FUNCTION_BLOCK PUBLIC FB_HeatingZone
VAR_INPUT
	mxEnableHeating 				: BOOL;
	mxReset							: BOOL;
	mxEmergency						: BOOL;
	mxDoorsOpened					: BOOL;
END_VAR
VAR_OUTPUT
	mxErrorInit						: BOOL;
	mxErrorStopInPos				: BOOL;
	Errors							: ST_HeatingZoneErrors;
END_VAR
VAR

	qxPWMOut1 AT%Q*					: BOOL;
	qxPWMOut2 AT%Q*					: BOOL;
	qxPWMOut3 AT%Q*					: BOOL;
	ixThermal AT%I*					: BOOL;
	
	FT_EnableHeating				:F_Trig;	

	FB_Heating_Controller			: FB_PIDCtrl;
	FB_PID							: FB_PID_CP;
	FB_PWM							: FB_CTRL_PWM_OUT;
	FB_Temperature					: FB_AnalogInPT100;
	RT_EmStop						: R_TRIG;
	FT_EmStop						: F_TRIG;
	ControlMode						: E_CTRL_MODE;
	RT_ActivateHeating				: R_TRIG;
	RT_TempError					: R_TRIG;
	
	T_TempBelowSetpoint				: TON;
	SR_TempBelowSetpoint			: SR;
	T_TempAboveSetpoint				: TON;
	SR_TempAboveSetpoint			: SR;
	T_TimeInAutomode				: TON;

	T_HeatingStarted				: TON;

	SR_PT100_Loose					: SR;
	SR_PT100_WireBreakActive		: SR;
	SR_PT100_HasWrongPosition		: SR;
	SR_PT100_NotInserted			: SR;
	SR_PT100_ConnectorNotConnected	: SR;
	SR_PT100_ResistorFound	: SR;
	
	T_PT100_CheckTemperatures		: TON;
	mxIncreasedTemperatureNonActive	: BOOL;
	mxNoIncreaseTemperatureActive	: BOOL;
	OldTemperature					: REAL;
	
	T_PT100_HasWrongPosition		: Ton;
	FT_ActivateHeating: F_TRIG;
	SR_PT100_EnabledZoneWithoutProperPt100: SR;
	SR_TemperatureWayTooHigh: SR;
	
	Setpoint 			 	: REAL;
	TemperatureDifference	: REAL;
	SetpointStep		 	: REAL;
	ActStepNr            	: INT;
	ActTempMemory 			: REAL;
	PIDsetpoint				: REAL;
	mxSetpointReached		: BOOL;
	T_TempAtSetpointDelayNextStep	: TON;
	RT_StartHeatingInSteps			: R_TRIG;
	HeatingInSteps					: BOOL;
	RT_StopHeatingInSteps: R_TRIG;
	RT_DoorOpened: R_TRIG;
	FT_DoorOpened: F_TRIG;
	RT_HeatingPIDON: R_TRIG;
	FT_HeatingPIDON: F_TRIG;
	RT_SetPointChanged: R_TRIG;
	OldSetpoint: REAL; 
	SR_TemperatureTooHighWarning: SR;
END_VAR
VAR_IN_OUT
	MachParameters					: ST_HeatingZone;
END_VAR

DetermineSetpoint();
Error();
Objects();

RT_ActivateHeating(CLK:=MachParameters.mxZoneActive);
T_HeatingStarted(IN:=, PT:=T#10M);

RT_HeatingPIDON(CLK:=FB_Heating_Controller.PID_ON);
FT_HeatingPIDON(CLK:=FB_Heating_Controller.PID_ON);

FB_Heating_Controller.PID_ON := mxEnableHeating AND MachParameters.mxZoneActive AND NOT mxEmergency AND NOT FB_Temperature.Error;

// Start heating "started" timer when heating switches on
IF RT_HeatingPIDON.Q THEN
	T_HeatingStarted.IN := TRUE;
END_IF

IF NOT FB_Heating_Controller.PID_ON THEN
	T_HeatingStarted.IN :=FALSE;
END_IF

// Autoreset the PWM controller when a error occures
IF FB_PWM.bError AND (ControlMode = eCTRL_MODE_ACTIVE) THEN
	Controlmode := eCTRL_MODE_RESET;
ELSE
	ControlMode := eCTRL_MODE_ACTIVE;
END_IF

OldSetpoint := MachParameters.PIDTempZone.SP_AUTO;

ACTION DetermineSetpoint:
// because of enormous overshoots, the setpoint of the PID is scaled up during startup
// and cut into smaller heating steps. For example when a 180 degree setpoint is set in the HMI
// And the number of warmingsteps is set to 10. The PID first gets a setpoint of: 180/10 * 1
// When the setpoint is reached the timer "SetpointReached" starts counting. When this timer
// is elapsed the next set is set into the PID -> 180/10 * 2.


RT_StartHeatingInSteps(CLK:=(FB_Heating_Controller.PV_EXT < MachParameters.LowLimitSP) AND RT_HeatingPIDON.Q);
RT_StopHeatingInSteps(CLK:=FT_HeatingPIDON.Q, Q=>);
T_TempAtSetpointDelayNextStep(IN:=mxSetpointReached, PT:=MachParameters.WaitTimeAfterStepReached);

// Interupt/stop heating in steps.
IF RT_StopHeatingInSteps.Q THEN HeatingInSteps:= FALSE; END_IF

//do this once when starting heating, determine setpoints.
IF RT_StartHeatingInSteps.q THEN
	HeatingInSteps := TRUE;
	
	TemperatureDifference := MachParameters.PIDTempZone.SP_AUTO_TOTAL - FB_Heating_Controller.PV_EXT;		// 160 = 180 - 20
	SetpointStep := TemperatureDifference / MachParameters.nrOfSteps;								// 16  = 160 / 10
	ActStepNr := 1;
	ActTempMemory := FB_Heating_Controller.PV_EXT;
	MachParameters.PIDTempZone.SP_AUTO := (ActStepNr * SetpointStep) + ActTempMemory;										// 1 * 16.0 + 20 =36.0 degree
END_IF

// When heating in steps is active the following code is active
IF HeatingInSteps THEN
		
	IF NOT mxSetpointReached AND (FB_Heating_Controller.PV_EXT >= MachParameters.PIDTempZone.SP_AUTO) THEN mxSetpointReached := TRUE; END_IF	
	
	IF T_TempAtSetpointDelayNextStep.q THEN
		
		mxSetpointReached := FALSE;
		
		IF ActStepNr < MachParameters.nrOfSteps THEN
			ActStepNr := ActStepNr + 1;
			MachParameters.PIDTempZone.SP_AUTO := (ActStepNr * SetpointStep) + ActTempMemory;			// 1 * 16.0 + 20 =36.0 degree
		ELSE
			ActStepNr := 1;
			HeatingInSteps := FALSE;
		END_IF;
			
	END_IF;
ELSE
	MachParameters.PIDTempZone.SP_AUTO := MachParameters.PIDTempZone.SP_AUTO_TOTAL;
END_IF;
END_ACTION

ACTION Error:
// FMEA errors .. //

//1 PT100 loose
SR_PT100_Loose(SET1:=SR_PT100_WireBreakActive.Q1 OR T_PT100_HasWrongPosition.Q OR SR_PT100_NotInserted.Q1, RESET:=mxReset, Q1=> );

//2 Wire break alarm (from terminal).
SR_PT100_WireBreakActive(Set1:= FB_Temperature.Wirebreak, Reset:=mxReset);

//3 check heating element zone, check if there is no difference in temperature over a x time while element is active
SR_PT100_HasWrongPosition(SET1:=NOT mxEmergency AND mxEnableHeating AND MachParameters.mxZoneActive AND mxNoIncreaseTemperatureActive  
AND (FB_Temperature.EngTempOut < (MachParameters.PIDTempZone.SP_AUTO - 40.0))  , Reset:=mxReset);

//4 check heating element zone, check if there is a difference in temperature over a x time while element is not
SR_PT100_NotInserted(SET1:=((NOT MachParameters.mxZoneActive) AND mxIncreasedTemperatureNonActive AND NOT T_HeatingStarted.Q), Reset:=mxReset); // testen!

// Other errors.. //
SR_PT100_EnabledZoneWithoutProperPt100(SET1:=(FB_Temperature.EngTempOut < 5.0) AND RT_ActivateHeating.Q, RESET:=mxReset );

IF (FB_Temperature.EngTempOut < 5.0) OR Errors.PT100_TemperatureAboveMaximum THEN
	MachParameters.mxZoneActive := FALSE;
END_IF

// Connector pt100 not connected: 100 ohm missing / pt100 , open loop.
SR_PT100_ConnectorNotConnected(SET1:=(FB_Temperature.EngTempOut > 750) , RESET:=mxReset);

// Is a warning now only, only alarm message in the HMI 
SR_TempBelowSetpoint(SET1:=T_TempBelowSetpoint.Q , RESET:= mxReset);
SR_TempAboveSetpoint(SET1:=T_TempAboveSetpoint.Q , RESET:= mxReset);

// Alarming timers
T_TempBelowSetpoint(IN:= mxEnableHeating AND MachParameters.mxZoneActive AND (FB_Temperature.EngTempOut < (MachParameters.PIDTempZone.SP_AUTO -15)), PT:=T#1M);
T_TempAboveSetpoint(IN:= mxEnableHeating AND MachParameters.mxZoneActive AND (FB_Temperature.EngTempOut > (MachParameters.PIDTempZone.SP_AUTO +15)), PT:=T#1M);

// reset the timer of the change in temperature when the setpoint is changed on the HMI
RT_SetPointChanged(CLK:= OldSetpoint <> MachParameters.PIDTempZone.SP_AUTO);

T_PT100_CheckTemperatures(IN:= NOT T_PT100_CheckTemperatures.Q AND FB_Heating_Controller.PID_ON AND NOT RT_SetPointChanged.Q, PT:=MachParameters.TimeErrorCheckinterval);
IF T_PT100_CheckTemperatures.Q THEN
	mxNoIncreaseTemperatureActive := mxIncreasedTemperatureNonActive := FALSE;
	mxNoIncreaseTemperatureActive := mxEnableHeating AND NOT (FB_Temperature.EngTempOut > (OldTemperature + MachParameters.TempErrorRaise));
	mxIncreasedTemperatureNonActive := mxEnableHeating AND (FB_Temperature.EngTempOut > (OldTemperature + MachParameters.TempErrorRaise));
	OldTemperature := FB_Temperature.EngTempOut;
END_IF

IF NOT FB_Heating_Controller.PID_ON THEN mxNoIncreaseTemperatureActive := mxIncreasedTemperatureNonActive := FALSE; END_IF

SR_TemperatureWayTooHigh(SET1:=(FB_Temperature.EngTempOut > 250) AND (FB_Temperature.EngTempOut < 300.0), RESET:=mxReset);
SR_TemperatureTooHighWarning(SET1:=(FB_Temperature.EngTempOut > 230) AND (FB_Temperature.EngTempOut < 300.0), RESET:=mxReset);


Errors.Thermal:= NOT ixThermal;
Errors.PT100_Loose := SR_PT100_Loose.Q1;
Errors.PT100_WireBreak := SR_PT100_WireBreakActive.Q1;	
Errors.PT100_HasWrongPosition := SR_PT100_HasWrongPosition.Q1;
Errors.PT100_NotInserted := SR_PT100_NotInserted.Q1;
Errors.PT100_ConnectorNotConnected := SR_PT100_ConnectorNotConnected.Q1;
Errors.PT100_TemperatureAboveMaximum := SR_TemperatureWayTooHigh.Q1;
Errors.PT100_TemperatureTooHighWarn := SR_TemperatureTooHighWarning.Q1;
 
(**********************************************************************************************************)
mxErrorStopinPos:= FALSE; 
mxErrorInit:= errors.PT100_TemperatureAboveMaximum OR Errors.PT100_Loose;// OR Errors.PT100_ConnectorNotConnected;
END_ACTION

ACTION Objects:
FB_Temperature(
	EngTempOut=> , 
	Error=> );

FB_PID(
	Enable:= FB_Heating_Controller.PID_ON, 
	Reset:= NOT FB_Heating_Controller.PID_ON, 
	TskCycleTime:= T#10MS, 
	CtrlCycleTime:= T#20MS);
	
FB_Heating_Controller(
	PID:= FB_PID,
	PV_EXT:= FB_Temperature.EngTempOut, 
	Parameters:= MachParameters.PIDTempZone);

FB_PWM(
	fPwmInput:= FB_Heating_Controller.OUT_PID, 
	eMode:= Controlmode, 
	bPwmOutBitPos=> , 
	bPwmOutBitNeg=> , 
	eState=> , 
	eErrorId=> , 
	bError=> , 
	stParams:= MachParameters.PWM_Parameters);
	
MachParameters.PWM_Parameters.tTaskCycleTime := T#10MS;
	
	(*Generate output when this mold heating is enabled*)
qxPWMOut1:= qxPWMOut2:= qxPWMOut3:= FB_PWM.bPwmOutBitPos AND MachParameters.mxZoneActive;
END_ACTION

END_FUNCTION_BLOCK

(* stored: Version 1.1.0.1, ProductVersion 3.1.4020.12
   POU FB_HeatingZone: Id {d65273e5-2158-4913-9345-73410858520a}, SpecialFunc None
   Action DetermineSetpoint: Id {fd7171c7-201a-4521-9c3d-8968f4828c63}
   Action Error: Id {b6863f51-4c4e-4c7d-93e8-ab62dbaf547f}
   Action Objects: Id {3afeabeb-9558-458b-8577-a9a8c0e82354} *)
